FUNCTION_BLOCK FB_TablePlace
VAR_INPUT
END_VAR
VAR_OUTPUT
END_VAR
VAR
	itfWorkingStation: I_WorkingStation;
	bRotationInterlock:BOOL;
	bRotationRequest: BOOL;
	bTableInPosition: BOOL;
	bWorkPermission: BOOL;
	bStationError: BOOL;
	udiErrorNumber: UDINT;
	bReleaseChange: BOOL;
END_VAR
VAR PERSISTENT
	stPlace: ST_TableBottlePlace;
	bMemOk : BOOL; 					//Sprawdzenie czy pamiec sie zinicjalizowala
END_VAR


bStationError := FALSE;
udiErrorNumber := 0;

IF prStateIsEmpty THEN
	stPlace.nBottleType:=nBottleTypes.none;
ELSIF NOT prStateIsEmpty AND stPlace.nBottleType=nBottleTypes.none THEN
	stPlace.nBottleType := nBottleTypes.first;
END_IF

IF itfWorkingStation = 0 THEN
	bRotationInterlock := TRUE;
	bRotationRequest := TRUE;
	bReleaseChange := TRUE;
ELSE
	bRotationInterlock := itfWorkingStation.prTableRotationInterlock;
	bRotationRequest := itfWorkingStation.prTableRotationRequest;
	bStationError := itfWorkingStation.prError;
	udiErrorNumber :=  itfWorkingStation.prErrorNumber;
	bReleaseChange := NOT itfWorkingStation.prWorkInProgress;
END_IF
bMemOk S= bTableInPosition;

IF NOT prStateIsNok AND NOT prStateIsDrawer THEN
	stPlace.byDetectionStatus := 0;
END_IF

METHOD mBottleAfterWeighing : BOOL
VAR_INPUT
END_VAR
IF prStateIsProcessing THEN
	stPlace.nState:=nTableBottlePlaceState.AfterWeighing;
END_IF;
mBottleAfterWeighing :=prStateIsAfterWeighing;
END_METHOD

METHOD mBottleBeforeWeighing : BOOL
VAR_INPUT
	nBottleType: nBottleTypes;
END_VAR
IF prStateIsEmpty AND  nBottleType <> nBottleTypes.none THEN
	stPlace.nState:=nTableBottlePlaceState.BeforeWeighing;
	stPlace.nBottleType:=nBottleType;
END_IF;
mBottleBeforeWeighing := prStateIsBeforeWeighing;
END_METHOD

METHOD mBottleDrawer : BOOL
VAR_INPUT
END_VAR
IF prStateIsNok THEN
	stPlace.nState:=nTableBottlePlaceState.Drawer;
END_IF;
mBottleDrawer := prStateIsDrawer;
END_METHOD

METHOD mBottleEmpty : BOOL
VAR_INPUT
END_VAR
IF prStateIsDrawer OR  prStateIsAfterWeighing  OR prStateIsTare THEN
	stPlace.nState:=nTableBottlePlaceState.Empty;
END_IF;
mBottleEmpty := prStateIsEmpty;
END_METHOD

METHOD mBottleNOK : BOOL
VAR_INPUT
END_VAR
IF prStateIsProcessing THEN
	stPlace.nState:=nTableBottlePlaceState.NOK;
END_IF;
mBottleNOK := prStateIsNOK;
END_METHOD

METHOD mBottleProcessing : BOOL
VAR_INPUT
END_VAR
IF prStateIsBeforeWeighing THEN
	stPlace.nState:=nTableBottlePlaceState.Processing;
END_IF;
mBottleProcessing := stPlace.nState=nTableBottlePlaceState.Processing;
END_METHOD

METHOD mBottleTare : BOOL
VAR_INPUT

END_VAR
IF prStateIsEmpty THEN
	stPlace.nState:=nTableBottlePlaceState.Tare;
END_IF;
mBottleTare := prStateIsTare;
END_METHOD

METHOD mClearWorkingStation : BOOL
VAR_INPUT
END_VAR
itfWorkingStation := 0;
END_METHOD

METHOD mDetectionStatus : BOOL
VAR_INPUT
	BitNum: SINT;
END_VAR
stPlace.byDetectionStatus:=DWORD_TO_BYTE(SETBIT32(stPlace.byDetectionStatus,BitNum));
END_METHOD

METHOD mErrorReset : BOOL
VAR_INPUT
END_VAR
IF itfWorkingStation <>0 THEN
	itfWorkingStation.mErrorReset();
END_IF
END_METHOD

PROPERTY pCurrentState : nTableBottlePlaceState
GET
pCurrentState:=stPlace.nState;
END_GET
END_PROPERTY

PROPERTY prBottleType : nBottleTypes
GET
prBottleType := stPlace.nBottleType;
END_GET
END_PROPERTY

{attribue 'monitoring':= call}
PROPERTY prCurrentPosition : USINT
GET
prCurrentPosition := stPlace.iCurrentPosition;
END_GET
SET
stPlace.iCurrentPosition := prCurrentPosition;
END_SET
END_PROPERTY

{attribue 'monitoring':= call}
PROPERTY prPlaceNumber : USINT
GET
prPlaceNumber := stPlace.iPlaceNumber;
END_GET
SET
stPlace.iPlaceNumber := prPlaceNumber;
END_SET
END_PROPERTY

PROPERTY prStateIsAfterWeighing : BOOL
GET
prStateIsAfterWeighing := stPlace.nState = nTableBottlePlaceState.AfterWeighing;
END_GET
END_PROPERTY

PROPERTY prStateIsBeforeWeighing : BOOL
GET
prStateIsBeforeWeighing := stPlace.nState = nTableBottlePlaceState.BeforeWeighing;
END_GET
END_PROPERTY

PROPERTY prStateIsDrawer : BOOL
GET
prStateIsDrawer := stPlace.nState = nTableBottlePlaceState.Drawer;
END_GET
END_PROPERTY

PROPERTY prStateIsEmpty : BOOL
GET
prStateIsEmpty := stPlace.nState = nTableBottlePlaceState.Empty;
END_GET
END_PROPERTY

PROPERTY prStateIsNOK : BOOL
GET
prStateIsNOK := stPlace.nState = nTableBottlePlaceState.NOK;
END_GET
END_PROPERTY

PROPERTY prStateIsProcessing : BOOL
GET
prStateIsProcessing := stPlace.nState = nTableBottlePlaceState.Processing;
END_GET
END_PROPERTY

PROPERTY prStateIsTare : BOOL
GET
prStateIsTare := stPlace.nState = nTableBottlePlaceState.Tare;
END_GET
END_PROPERTY

PROPERTY prTableInPosition : BOOL
GET
prTableInPosition:= bTableInPosition;
END_GET
SET
bTableInPosition:= prTableInPosition;
END_SET
END_PROPERTY

{attribue 'monitoring':= call}
PROPERTY prTableRotationInterlock : BOOL
GET
prTableRotationInterlock:=bRotationInterlock;
END_GET
END_PROPERTY

{attribue 'monitoring':= call}
PROPERTY prTableRotationRequest : BOOL
GET
prTableRotationRequest:=bRotationRequest;
END_GET
END_PROPERTY

{attribue 'monitoring':= call}
PROPERTY pWorkingStation : I_WorkingStation
GET
pWorkingStation:=itfWorkingStation;
END_GET
SET
itfWorkingStation:=pWorkingStation;
END_SET
END_PROPERTY

END_FUNCTION_BLOCK

(* stored: Version 1.1.0.1, ProductVersion 3.1.4024.15
   POU FB_TablePlace: Id {265b384e-c169-4e44-874d-ccc78b9ed3f4}, SpecialFunc None
   Method mBottleAfterWeighing: Id {9720bd92-134b-4b68-80c2-6a2cc402d47b}
   Method mBottleBeforeWeighing: Id {0e51995b-61d3-4d5c-9d79-3d4ce30af29a}
   Method mBottleDrawer: Id {f7231045-de72-4f36-a4fc-f1a29dee7baa}
   Method mBottleEmpty: Id {ca40ada9-4135-4273-bf5c-545dda9a8893}
   Method mBottleNOK: Id {8efc58f1-e306-405d-8f2e-c3151afc8a3a}
   Method mBottleProcessing: Id {78fece03-d3c1-4513-b438-a2dda4dd1d85}
   Method mBottleTare: Id {f8ef4a5d-c4ba-47a2-8172-bcea1faf3417}
   Method mClearWorkingStation: Id {596c1c0d-7109-4b79-96a8-9dcefd06f95c}
   Method mDetectionStatus: Id {4ea23455-2941-46cb-a99a-b0cd25f99f28}
   Method mErrorReset: Id {f81092d1-2e8f-4f01-8d86-b3405151cafb}
   Property pCurrentState: Id {d551517b-b62f-46c5-9d0d-b7f371e0d162}
   Get Get: Id {4c6e54f6-27c3-4729-a897-f5ba85736deb}
   Property prBottleType: Id {00e4f692-a5ec-473b-9b55-a05c993e152b}
   Get Get: Id {f25e6ee1-1ce5-4dd6-b172-15f7dd3acf4b}
   Property prCurrentPosition: Id {a591398c-db6a-47a5-a1b9-1fc16684ff4f}
   Get Get: Id {1aa8cdb1-493e-4214-b67a-9d66cba99e49}
   Set Set: Id {98f3d7e6-effe-4813-a325-574167bd8b3d}
   Property prPlaceNumber: Id {7935c5e2-73d5-45fc-b6fd-9b8d28dbb8a1}
   Get Get: Id {82ddc4e6-e54d-4d5d-999c-fb8a41ab6951}
   Set Set: Id {7adaf66a-cc0e-4f34-a3ee-212285cd5fc5}
   Property prStateIsAfterWeighing: Id {ebec9ad5-df36-4242-88ed-d5c1d697457e}
   Get Get: Id {575bcb67-28b6-48cd-87b4-1c0e88c9ec46}
   Property prStateIsBeforeWeighing: Id {481ad8af-6a50-49bb-aca4-2a9f22a0e63f}
   Get Get: Id {6f2377f6-3f48-4441-aebe-9ea63c399cdb}
   Property prStateIsDrawer: Id {3e6346b5-9e6b-4151-8761-38edf1f53eef}
   Get Get: Id {f080b430-b234-49c5-b0d3-77d1bcf308ff}
   Property prStateIsEmpty: Id {1ee73aaa-35be-4134-bcd5-1ba73af556b8}
   Get Get: Id {aaccb4bb-77bb-4e85-945a-35d2b23bde3a}
   Property prStateIsNOK: Id {5c9ec95c-c0f5-4133-ab9e-4e8c2e271bfa}
   Get Get: Id {8c142683-8479-46ca-8ee4-398522b8b640}
   Property prStateIsProcessing: Id {fbf96f1f-e4c1-44c9-9f56-2a2fdadc3610}
   Get Get: Id {b206eed4-5a9c-4058-964a-88ec02de02dc}
   Property prStateIsTare: Id {82446558-3544-4623-9d90-87e48767d493}
   Get Get: Id {9dcba566-5318-4dab-afe0-a3e22e42d5c4}
   Property prTableInPosition: Id {e89e4850-00f9-481f-8561-f2be797aad18}
   Get Get: Id {0b833c6d-0098-4be4-b16c-f8cbee68f653}
   Set Set: Id {5a6baea0-075a-4e4f-92cf-9ed15f17ea2f}
   Property prTableRotationInterlock: Id {294c7375-f490-4e19-8180-0f73a52a88e1}
   Get Get: Id {6f7f66c3-b6d2-460f-9b0e-c2638fe9ae18}
   Property prTableRotationRequest: Id {7c83dcbf-0e28-497b-9f6e-109f400d7f6c}
   Get Get: Id {a27aa4c2-9571-4e96-bf1a-f7e87f67c113}
   Property pWorkingStation: Id {a880ebf4-8ac0-4f02-aadc-ac1b7bc377ec}
   Get Get: Id {fe8ca71b-91c3-405b-b7fe-d8e6f8ad29ff}
   Set Set: Id {30faeb23-cb76-460c-9989-0b0d18edc710} *)
